FUNCTION_BLOCK T_ClearGroupCountEqualsZeroCompareEqualsFalse EXTENDS T_UnitTestBase
VAR
  list : T_ComponentsCollection(10);
  newComponent : ARRAY [1..5] OF T_Component;
  afterCountActual, afterCountExpected : UINT;
  beforeCountActual, beforeCountExpected : UINT;
  beforeActual, beforeExpected : I_ComponentBase;
  afterActual, afterExpected : I_ComponentBase;
 beforeResult, afterResult : BOOL;
END_VAR

// Arrange
list.AddComponent(newComponent[1]);
list.AddComponent(newComponent[2]);
list.AddComponent(newComponent[3]);
list.AddComponent(newComponent[4]);

// first test before running clear
beforeExpected := newComponent[1];
__QUERYINTERFACE(list._items[0], beforeActual);
beforeResult := beforeExpected = beforeActual;

Assertion.AssertEquals_BOOL(TRUE, beforeResult, 'item 0 = list.AddComponent()');
Assertion.AssertEquals_UDINT(4, list.Count, 'list.Count = 4');

//Act
list.ClearGroup();

//Assert 
afterExpected := newComponent[1];
__QUERYINTERFACE(list._items[0], afterActual);
afterResult := afterExpected <> afterActual;
Assertion.AssertEquals_BOOL(TRUE, beforeResult, 'afterResult := afterExpected <> afterActual;');

afterCountActual := list.Count;
afterCountExpected := 0;
Assertion.AssertEquals_UDINT(afterCountExpected, afterCountActual, 'afterCountActul = 0');

TestFinished();

END_FUNCTION_BLOCK

(* stored: Version 1.1.0.1, ProductVersion 3.1.4024.12
   POU T_ClearGroupCountEqualsZeroCompareEqualsFalse: Id {a5ac6aae-d815-4031-8abd-dd6bd35c8542}, SpecialFunc None *)
